(* LS Electric XG5000 project: 20230520 *)
(* PLC LSPLC *)
VAR_GLOBAL
    T1 : TP;
    스위치 AT %MX0 : BOOL := 1;
END_VAR

PROGRAM NewProgram (* task: 스캔 프로그램 *)
VAR
    cnt : CTU_INT;
    input AT %IW0.1.0 : INT;
    inputTime : TIME;
    INST : CTD_INT;
    INST1 : CTD_INT;
    INST2 : CTD_INT;
    str1 : STRING;
    str2 : STRING;
    스위치1 AT %MX1 : BOOL;
END_VAR
VAR_EXTERNAL
    T1 : TP;
    스위치 : BOOL; (* AT %MX0 *)
END_VAR

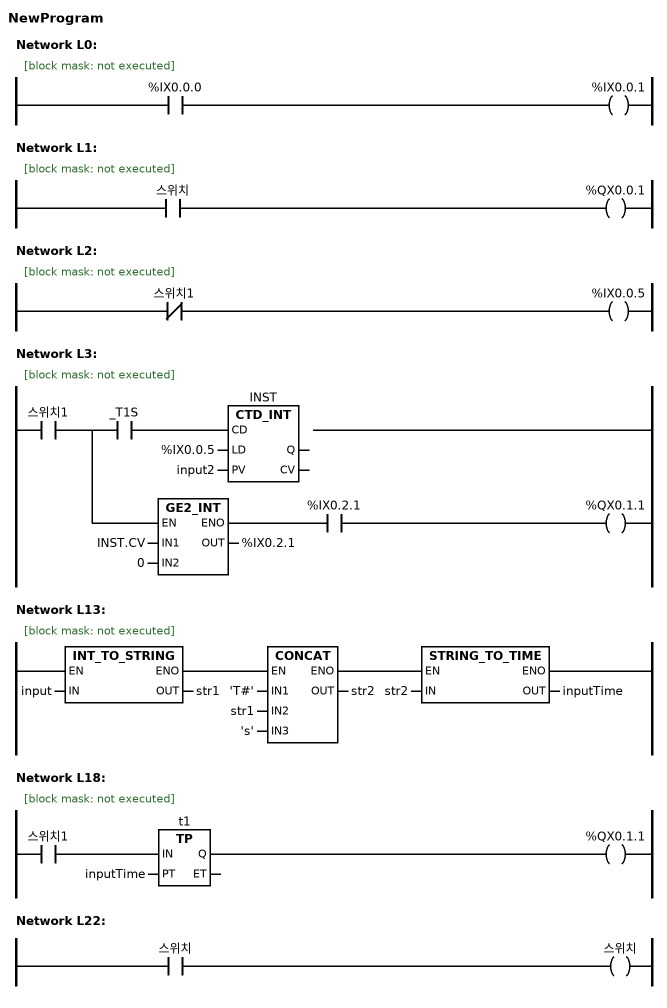
(* Rung L0 is block-masked: not executed *)
// %IX0.0.1 := %IX0.0.0;
(* Rung L1 is block-masked: not executed *)
// %QX0.0.1 := 스위치;
(* Rung L2 is block-masked: not executed *)
// %IX0.0.5 := NOT 스위치1;
(* Rung L3 is block-masked: not executed *)
// INST(CD := 스위치1 AND _T1S, LD := %IX0.0.5, PV := input2);
// IF 스위치1 THEN %IX0.2.1 := GE2_INT(INST.CV, 0); END_IF;
// %QX0.1.1 := 스위치1 AND %IX0.2.1;
(* Rung L13 is block-masked: not executed *)
// str1 := INT_TO_STRING(input);
// str2 := CONCAT('T#', str1, 's');
// inputTime := STRING_TO_TIME(str2);
(* Rung L18 is block-masked: not executed *)
// t1(IN := 스위치1, PT := inputTime);
// %QX0.1.1 := t1.Q;
(* Rung L22 *)
스위치 := 스위치;
END_PROGRAM